{attribute 'qualified_only'}
VAR_GLOBAL
	bRunningLight : BOOL;
	fCylinderStroke : REAL;
	fCylinderVelocity : REAL;
	fTimeInSeconds : REAL;
END_VAR

(* stored: Version 1.1.0.1, ProductVersion 3.1.4024.10
   GVL output: Id {50514818-2454-4f82-b3b0-4985051ea887} *)
